// SIMATIC STEP 7 (V5.x) project tp7
// CPU: CPU 312 IFM
// station: Matériel
// station: SIMATIC 300(1)
// station: P_ADR_BUS
// station: ISA_LOCAL_ADR_BUS
// program: Programme S7(6)

SYMBOL_TABLE
"DP_SEND"	FC 1	FC 1	// DP SEND
"DP_RECV"	FC 2	FC 2	// DP RECEIVE
END_SYMBOL_TABLE

// FC 1: know-how protected block, not included

// FC 2: know-how protected block, not included

ORGANIZATION_BLOCK OB 1
TITLE = "Main Program Sweep (Cycle)"
VERSION : 0.1
VAR_TEMP
  OB1_EV_CLASS : BYTE ;	//Bits 0-3 = 1 (Coming event), Bits 4-7 = 1 (Event class 1)
  OB1_SCAN_1 : BYTE ;	//1 (Cold restart scan 1 of OB 1), 3 (Scan 2-n of OB 1)
  OB1_PRIORITY : BYTE ;	//Priority of OB Execution
  OB1_OB_NUMBR : BYTE ;	//1 (Organization block 1, OB1)
  OB1_RESERVED_1 : BYTE ;	//Reserved for system
  OB1_RESERVED_2 : BYTE ;	//Reserved for system
  OB1_PREV_CYCLE : INT ;	//Cycle time of previous OB1 scan (milliseconds)
  OB1_MIN_CYCLE : INT ;	//Minimum cycle time of OB1 (milliseconds)
  OB1_MAX_CYCLE : INT ;	//Maximum cycle time of OB1 (milliseconds)
  OB1_DATE_TIME : DATE_AND_TIME ;	//Date and time OB1 started
END_VAR
BEGIN
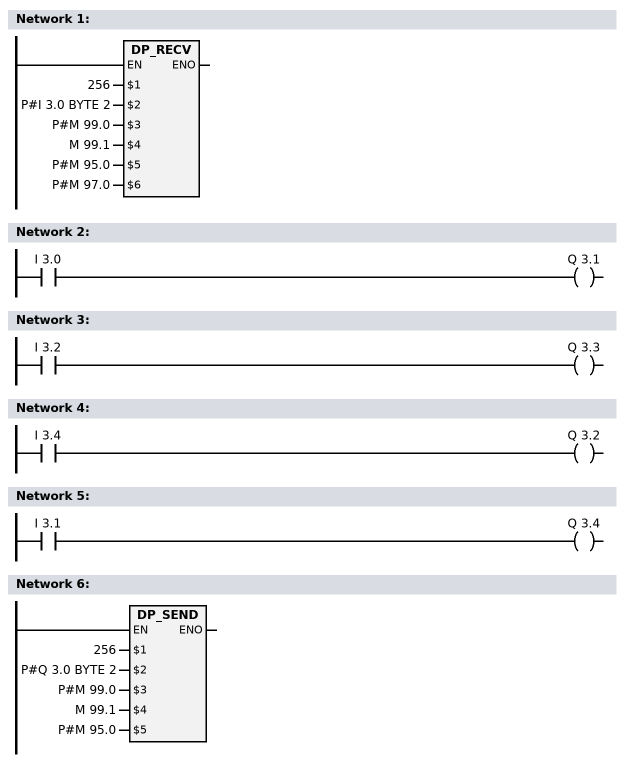
NETWORK
TITLE =
      CALL  "DP_RECV" (
           $1                       := 256,
           $2                       := P#I 3.0 BYTE 2,
           $3                       := P#M 99.0,
           $4                       := M 99.1,
           $5                       := P#M 95.0,
           $6                       := P#M 97.0);
      NOP   0;
NETWORK
TITLE =
      A     I 3.0;
      =     Q 3.1;
NETWORK
TITLE =
      A     I 3.2;
      =     Q 3.3;
NETWORK
TITLE =
      A     I 3.4;
      =     Q 3.2;
NETWORK
TITLE =
      A     I 3.1;
      =     Q 3.4;
NETWORK
TITLE =
      CALL  "DP_SEND" (
           $1                       := 256,
           $2                       := P#Q 3.0 BYTE 2,
           $3                       := P#M 99.0,
           $4                       := M 99.1,
           $5                       := P#M 95.0);
      NOP   0;
END_ORGANIZATION_BLOCK
